# EPICS substitutions: evrMrmApp/Db/evr-vme-300.substitutions
# Record set for a VME-EVRRF-230
#
# Macros:
#  EVR = Card name (same as mrmEvrSetupVME())
#  SYS = System name (ie SR-TM)
#

file "evr-base.template"
{pattern
{ SYS,      EVR,     EVNT1HZ}
{"$(SYS)", "$(EVR)", 125}
}

file "sfp.template"
{
{SYS="$(SYS)", EVR="$(EVR)", ID="0"}
}

file "flash.template"
{
{SYS="$(SYS)", EVG="$(EVR)"}
}

file "evr-prescaler.template"
{pattern
{ SYS,      EVR,     ID, MAX}
{"$(SYS)", "$(EVR)", 0, "0xffffffff"}
{"$(SYS)", "$(EVR)", 1, "0xffffffff"}
{"$(SYS)", "$(EVR)", 2, "0xffffffff"}
{"$(SYS)", "$(EVR)", 3, "0xffffffff"}
{"$(SYS)", "$(EVR)", 4, "0xffffffff"}
{"$(SYS)", "$(EVR)", 5, "0xffffffff"}
{"$(SYS)", "$(EVR)", 6, "0xffffffff"}
{"$(SYS)", "$(EVR)", 7, "0xffffffff"}
}

# Pulse generators w/o a prescaler set NOPS=1
# TODO this form factor has pul0 - pul23
file "evr-pulser.template"
{pattern
{ SYS,      EVR,     ID,  DMAX,       WMAX,          PMAX,  NOPS}
{"$(SYS)", "$(EVR)", 0,  "0xffffffff", "0xffffffff", "0xffff", 0}
{"$(SYS)", "$(EVR)", 1,  "0xffffffff", "0xffffffff", "0xffff", 0}
{"$(SYS)", "$(EVR)", 2,  "0xffffffff", "0xffffffff", "0xffff", 0}
{"$(SYS)", "$(EVR)", 3,  "0xffffffff", "0xffffffff", "0xffff", 0}
{"$(SYS)", "$(EVR)", 4,  "0xffffffff", "0xffff",     "1",      1}
{"$(SYS)", "$(EVR)", 5,  "0xffffffff", "0xffff",     "1",      1}
{"$(SYS)", "$(EVR)", 6,  "0xffffffff", "0xffff",     "1",      1}
{"$(SYS)", "$(EVR)", 7,  "0xffffffff", "0xffff",     "1",      1}
{"$(SYS)", "$(EVR)", 8,  "0xffffffff", "0xffff",     "1",      1}
{"$(SYS)", "$(EVR)", 9,  "0xffffffff", "0xffff",     "1",      1}
{"$(SYS)", "$(EVR)", 10, "0xffffffff", "0xffff",     "1",      1}
{"$(SYS)", "$(EVR)", 11, "0xffffffff", "0xffff",     "1",      1}
{"$(SYS)", "$(EVR)", 12, "0xffffffff", "0xffff",     "1",      1}
{"$(SYS)", "$(EVR)", 13, "0xffffffff", "0xffff",     "1",      1}
{"$(SYS)", "$(EVR)", 14, "0xffffffff", "0xffff",     "1",      1}
{"$(SYS)", "$(EVR)", 15, "0xffffffff", "0xffff",     "1",      1}
{"$(SYS)", "$(EVR)", 16, "0xffffffff", "0xffff",     "1",      1}
{"$(SYS)", "$(EVR)", 17, "0xffffffff", "0xffff",     "1",      1}
{"$(SYS)", "$(EVR)", 18, "0xffffffff", "0xffff",     "1",      1}
{"$(SYS)", "$(EVR)", 19, "0xffffffff", "0xffff",     "1",      1}
{"$(SYS)", "$(EVR)", 20, "0xffffffff", "0xffff",     "1",      1}
{"$(SYS)", "$(EVR)", 21, "0xffffffff", "0xffff",     "1",      1}
{"$(SYS)", "$(EVR)", 22, "0xffffffff", "0xffff",     "1",      1}
{"$(SYS)", "$(EVR)", 23, "0xffffffff", "0xffff",     "1",      1}

{"$(SYS)", "$(EVR)", 24, "0xffffffff", "0xffff",     "1",      1}
{"$(SYS)", "$(EVR)", 25, "0xffffffff", "0xffff",     "1",      1}
{"$(SYS)", "$(EVR)", 26, "0xffffffff", "0xffff",     "1",      1}
{"$(SYS)", "$(EVR)", 27, "0xffffffff", "0xffff",     "1",      1}
{"$(SYS)", "$(EVR)", 28, "0xffffffff", "0xffff",     "1",      1}
{"$(SYS)", "$(EVR)", 29, "0xffffffff", "0xffff",     "1",      1}
{"$(SYS)", "$(EVR)", 30, "0xffffffff", "0xffff",     "1",      1}
{"$(SYS)", "$(EVR)", 31, "0xffffffff", "0xffff",     "1",      1}
}

## Form factor specific

file "evr-in.template"
{pattern
{ SYS,      EVR,     ID,  DESC}
{"$(SYS)", "$(EVR)", 0,  "IN0 (TTL)"}
{"$(SYS)", "$(EVR)", 1,  "IN1 (TTL)"}
}

## TODO add 16 transition board inputs

file "evr-out.template"
{pattern
{ SYS,      EVR,      OBJ,    		 	ID,   DESC}
{"$(SYS)", "$(EVR)", "FrontUnivOut", 	0,   "UNIV0"}
{"$(SYS)", "$(EVR)", "FrontUnivOut", 	1,   "UNIV1"}
{"$(SYS)", "$(EVR)", "FrontUnivOut", 	2,   "UNIV2"}
{"$(SYS)", "$(EVR)", "FrontUnivOut", 	3,   "UNIV3"}
{"$(SYS)", "$(EVR)", "FrontUnivOut", 	4,   "UNIV4"}
{"$(SYS)", "$(EVR)", "FrontUnivOut", 	5,   "UNIV5"}
{"$(SYS)", "$(EVR)", "FrontUnivOut", 	6,   "UNIV6 (CML)"}
{"$(SYS)", "$(EVR)", "FrontUnivOut", 	7,   "UNIV7 (CML)"}
{"$(SYS)", "$(EVR)", "FrontUnivOut", 	8,   "UNIV8 (CML)"}
{"$(SYS)", "$(EVR)", "FrontUnivOut", 	9,   "UNIV9 (CML)"}
{"$(SYS)", "$(EVR)", "RearUniv", 		0,   "TRANSITION 0"}
{"$(SYS)", "$(EVR)", "RearUniv", 		1,   "TRANSITION 1"}
{"$(SYS)", "$(EVR)", "RearUniv", 		2,   "TRANSITION 2"}
{"$(SYS)", "$(EVR)", "RearUniv", 		3,   "TRANSITION 3"}
{"$(SYS)", "$(EVR)", "RearUniv", 		4,   "TRANSITION 4"}
{"$(SYS)", "$(EVR)", "RearUniv", 		5,   "TRANSITION 5"}
{"$(SYS)", "$(EVR)", "RearUniv", 		6,   "TRANSITION 6"}
{"$(SYS)", "$(EVR)", "RearUniv", 		7,   "TRANSITION 7"}
{"$(SYS)", "$(EVR)", "RearUniv", 		8,   "TRANSITION 8"}
{"$(SYS)", "$(EVR)", "RearUniv", 		9,   "TRANSITION 9"}
{"$(SYS)", "$(EVR)", "RearUniv", 		10,  "TRANSITION 10"}
{"$(SYS)", "$(EVR)", "RearUniv", 		11,  "TRANSITION 11"}
{"$(SYS)", "$(EVR)", "RearUniv", 		12,  "TRANSITION 12"}
{"$(SYS)", "$(EVR)", "RearUniv", 		13,  "TRANSITION 13"}
{"$(SYS)", "$(EVR)", "RearUniv", 		14,  "TRANSITION 14"}
{"$(SYS)", "$(EVR)", "RearUniv", 		15,  "TRANSITION 15"}
}

file "evr-cml.template"
{pattern
{ SYS,      EVR,     ID, NBIT, MAX   }
{"$(SYS)", "$(EVR)", 0,  40,   81880 }
{"$(SYS)", "$(EVR)", 1,  40,   81880 }
{"$(SYS)", "$(EVR)", 2,  40,   81880 }
{"$(SYS)", "$(EVR)", 3,  40,   81880 }
}

file "evr-pulserMap-dbus.template"
{pattern
{ SYS,      EVR,     ID}
{"$(SYS)", "$(EVR)", 0}
{"$(SYS)", "$(EVR)", 1}
{"$(SYS)", "$(EVR)", 2}
{"$(SYS)", "$(EVR)", 3}
{"$(SYS)", "$(EVR)", 4}
{"$(SYS)", "$(EVR)", 5}
{"$(SYS)", "$(EVR)", 6}
{"$(SYS)", "$(EVR)", 7}
}
